//{attribute 'qualified_only'}
{attribute 'strict'}
TYPE E_FileGenerateStep :
(
	init := 0
	,Open
	,Write
	,Close
);
END_TYPE

(* stored: Version 1.1.0.1, ProductVersion 3.1.4024.6
   DUT E_FileGenerateStep: Id {507c61d1-35b6-475e-be50-a59705918ac2} *)
